Yaskawa INFORM job: R2_W31(0,0)_MP_OK.JBI

/JOB
//NAME R2_W31(0,0)_MP_OK
///FOLDERNAME MP_TEST
//POS
///NPOS 63,63,0,3,0,0
///TOOL 0
///POSTYPE PULSE
///PULSE
C00000=102126,18825,-41470,-65608,62226,36597
C00001=120339,23079,-19532,-81795,45939,24488
C00002=122189,67376,29099,-89357,43616,27152
C00003=121004,73460,34134,-89018,42790,27107
C00004=120543,75972,36286,-88933,42467,27118
C00005=120547,77449,38075,-89311,42453,27349
C00006=120543,75972,36286,-88933,42467,27118
C00007=123298,89224,41655,-76600,55308,25879
C00008=122969,89182,41601,-76463,55094,25842
C00009=119753,75938,36143,-88643,41920,27049
C00010=122777,93473,61536,-103228,51808,35130
C00011=122777,93480,60664,-102807,51709,34821
C00012=122056,93390,61432,-103190,51294,35173
C00013=122567,91090,59506,-103202,51654,35130
C00014=123870,85634,55138,-103330,52596,35092
C00015=122431,75509,15675,-42518,64116,27745
C00016=120732,80304,21747,-41899,62444,27757
C00017=114671,71267,10742,-25968,56507,20900
C00018=114705,72531,12271,-26076,56252,20980
C00019=120070,82309,24307,-41679,61753,27775
C00020=119168,83067,23974,-40915,61831,27344
C00021=118706,83060,23966,-40627,61642,27221
C00022=123924,66248,9738,-82632,66113,-4047
C00023=107346,82155,44839,-154040,38328,-19284
C00024=107345,82085,44753,-154030,38313,-19290
C00025=107345,82076,44742,-154029,38311,-19290
C00026=105787,83979,48622,-160749,39408,-16514
C00027=107604,79582,41685,-153491,37881,-19627
C00028=107224,79409,41473,-153690,37712,-19470
C00029=105695,84345,57528,-163375,44143,-15284
C00030=105497,78624,56137,-164243,46040,-14757
C00031=105622,85248,64438,-164704,47679,-14459
C00032=107258,82886,61095,-119534,27741,-31091
C00033=106881,82684,60844,-119663,27474,-31013
C00034=105608,84808,47557,-160750,38172,-16883
C00035=106033,81368,44275,-160360,38056,-17159
C00036=105627,84087,47624,-160957,38555,-16773
C00037=107258,82806,60996,-119500,27732,-31108
C00038=106881,82604,60746,-119629,27464,-31030
C00039=105638,83945,56237,-163246,43560,-15407
C00040=105896,77477,52492,-163460,44578,-15292
C00041=105548,77217,41300,-160829,38199,-16836
C00042=105602,86513,40989,-157937,33682,-18444
C00043=107257,82726,60897,-119467,27722,-31125
C00044=106880,82524,60648,-119596,27455,-31047
C00045=105576,86195,41386,-158222,34042,-18287
C00046=105951,77674,28448,-155386,30954,-19846
C00047=105669,83350,42706,-159534,36136,-17580
C00048=105566,85122,44827,-159825,36466,-17406
C00049=107256,82646,60799,-119433,27713,-31142
C00050=106879,82445,60550,-119562,27446,-31064
C00051=109596,83788,36714,-137443,34940,-24236
C00052=110362,76235,26997,-134418,33961,-25844
C00053=110080,77212,36112,-139665,37329,-22921
C00054=109684,81187,41006,-140766,37887,-22236
C00055=107256,82566,60701,-119400,27704,-31159
C00056=106879,82365,60452,-119529,27437,-31081
C00057=109652,80299,44547,-142980,39863,-20946
C00058=109696,79496,48486,-145056,42085,-19714
C00059=111201,59852,25009,-141057,39445,-22245
C00060=111201,74974,83144,-154603,62561,-12728
C00061=48826,-12478,-44952,-111799,21990,-32460
C00062=48826,-14822,-37600,-124145,24456,-26472
BC00000=73931,307281,837779
BC00001=58622,333960,766983
BC00002=57127,336566,760067
BC00003=57127,336566,760067
BC00004=57127,336566,760067
BC00005=57127,336566,760067
BC00006=57127,336566,760067
BC00007=57127,336566,760067
BC00008=57127,336566,760067
BC00009=57127,336566,760067
BC00010=57127,336566,760067
BC00011=57127,336566,760067
BC00012=57127,336566,760067
BC00013=57127,336566,760067
BC00014=57127,336566,760067
BC00015=59666,336099,348167
BC00016=59666,336099,348167
BC00017=59666,336099,348167
BC00018=59666,336099,348167
BC00019=59666,336099,348167
BC00020=59666,336099,348167
BC00021=59666,336099,348167
BC00022=47019,346669,514312
BC00023=32533,358775,704605
BC00024=32553,329698,597054
BC00025=36828,324081,608367
BC00026=36826,324083,608359
BC00027=38538,321835,612892
BC00028=38538,321835,612892
BC00029=36828,324081,608366
BC00030=36828,324081,608367
BC00031=36828,324081,608367
BC00032=21216,345689,787864
BC00033=21216,345689,787864
BC00034=36828,324081,443157
BC00035=36828,324081,407024
BC00036=36828,324081,407024
BC00037=21238,345779,684592
BC00038=21238,345779,684592
BC00039=36828,324081,407024
BC00040=36828,324081,407024
BC00041=36828,324081,313069
BC00042=36828,324081,237457
BC00043=21261,345868,581320
BC00044=21261,345868,581320
BC00045=36828,324081,188211
BC00046=36828,324081,174572
BC00047=36828,324081,174572
BC00048=36828,324081,174572
BC00049=21284,345957,478048
BC00050=21284,345957,478048
BC00051=36828,323509,113964
BC00052=36828,323494,112363
BC00053=36827,323494,112362
BC00054=36828,323494,112363
BC00055=21306,346047,374776
BC00056=21306,346047,374776
BC00057=36828,323494,112363
BC00058=36828,323494,112363
BC00059=36828,323494,112363
BC00060=36828,323494,367967
BC00061=36828,323494,367967
BC00062=36828,323494,1041515
///POSTYPE BASE
///RECTAN
///RCONF 0,0,0,0,0,0,0,0,0,0,0,0,0,0,0,0,0,0,0,0,0,0,0,0
P00006=0.222,-3.123,-1.508,0.0000,0.0000,0.0000
P00021=-0.225,-6.128,-0.405,0.0000,0.0000,0.0000
P00022=0.222,-3.123,-1.508,0.0000,0.0000,0.0000
//INST
///DATE 2023/11/16 10:45
///ATTR SC,RW
///GROUP1 RB1,BS1
NOP
SFTOF
'r2_W31(0,0)
'Path S948 (for W950)
SFTOF
MOVJ C00000 BC00000 VJ=20.00
MOVJ C00001 BC00001 VJ=20.00
MOVJ C00002 BC00002 VJ=20.00
MOVL C00003 BC00003 V=100.0
MOVL C00004 BC00004 V=60.0
REFP 3 C00005 BC00005
CALL JOB:SEARCH-R1
SET P021 P006
SFTON P021
MOVL C00006 BC00006 V=60.0
MOVL C00007 BC00007 V=60.0
REFP 3 C00008 BC00008
CALL JOB:SEARCH-R1
SET P021 P006
SFTON P021
MOVL C00009 BC00009 V=60.0
MOVL C00010 BC00010 V=60.0
REFP 3 C00011 BC00011
CALL JOB:SEARCH-R1
SET P021 P006
SFTON P021
MOVL C00012 BC00012 V=60.0
MOVL C00013 BC00013 V=100.0
MOVL C00014 BC00014 V=100.0
'Path S949 (for W950)
SFTOF
MOVJ C00015 BC00015 VJ=20.00
MOVL C00016 BC00016 V=100.0
MOVL C00017 BC00017 V=60.0
REFP 3 C00018 BC00018
CALL JOB:SEARCH-R1
SET P022 P006
SFTON P022
MOVL C00019 BC00019 V=60.0
MOVL C00020 BC00020 V=60.0
REFP 3 C00021 BC00021
CALL JOB:SEARCH-R1
SET P022 P006
SFTON P022
'Path W950
SFTOF
MOVJ C00022 BC00022 VJ=20.00
MOVJ C00023 BC00023 VJ=20.00
SFTON P021
MOVJ C00024 BC00024 VJ=20.00
MOVL C00025 BC00025 V=100.0
MOVL C00026 BC00026 V=100.0 PL=0
REFP 1 C00027 BC00027
REFP 2 C00028 BC00028
MACRO1 MJ#(0) ARGF10
ARCON
MOVL C00029 BC00029 V=9.2
ARCOF
MOVL C00030 BC00030 V=100.0
MOVL C00031 BC00031 V=100.0 PL=0
REFP 1 C00032 BC00032
REFP 2 C00033 BC00033
MACRO1 MJ#(0) ARGF10
ARCON
MOVL C00034 BC00034 V=9.2
ARCOF
MOVL C00035 BC00035 V=100.0
MOVL C00036 BC00036 V=100.0 PL=0
REFP 1 C00037 BC00037
REFP 2 C00038 BC00038
MACRO1 MJ#(0) ARGF0
ARCON
MOVL C00039 BC00039 V=9.2
ARCOF
MOVL C00040 BC00040 V=100.0
MOVL C00041 BC00041 V=100.0
SFTON P022
MOVL C00042 BC00042 V=100.0 PL=0
REFP 1 C00043 BC00043
REFP 2 C00044 BC00044
MACRO1 MJ#(0) ARGF10
ARCON
MOVL C00045 BC00045 V=9.2
ARCOF
MOVL C00046 BC00046 V=100.0
MOVL C00047 BC00047 V=100.0
MOVL C00048 BC00048 V=100.0 PL=0
REFP 1 C00049 BC00049
REFP 2 C00050 BC00050
MACRO1 MJ#(0) ARGF10
ARCON
MOVL C00051 BC00051 V=9.2
ARCOF
MOVL C00052 BC00052 V=100.0
MOVL C00053 BC00053 V=100.0
MOVL C00054 BC00054 V=100.0 PL=0
REFP 1 C00055 BC00055
REFP 2 C00056 BC00056
MACRO1 MJ#(0) ARGF10
ARCON
MOVL C00057 BC00057 V=9.2
MOVL C00058 BC00058 V=9.2
ARCOF
MOVL C00059 BC00059 V=100.0
MOVL C00060 BC00060 V=100.0
MOVL C00061 BC00061 V=100.0
SFTOF
MOVJ C00062 BC00062 VJ=20.00
END
